// TIA Portal V18 export
DATA_BLOCK "Function Flush"   // DB47
{ S7_Optimized_Access := 'TRUE' }
VERSION : 0.1
// stored: AutoNumber true, DBAccessibleFromOPCUA true, IsOnlyStoredInLoadMemory false, IsRetainMemResEnabled false, IsWriteProtectedInAS false, MemoryReserve 100
   VAR RETAIN
      Selection : Int;
      "Input A" : Struct
         "set qty" : Real;
         "set flowrate" : Real;
         "Set time" : Int;
         "set time IN MINUTES" : Real;
         "set time in sec" : DInt;
      END_STRUCT;
      "Input B" : Struct
         "set qty" : Real;
         "set flowrate" : Real;
         "Set time" : Int;
         "set time IN MINUTES" : Real;
         "set time in sec" : DInt;
      END_STRUCT;
   END_VAR
   VAR
      "Control A" : Struct
         "Start flushing" : Bool;
         "Stop Flushing" : Bool;
         "flush running" : Bool;
         "flush Completed" : Bool;
      END_STRUCT;
      "Control B" : Struct
         "Start flushing" : Bool;
         "Stop Flushing" : Bool;
         "flush running" : Bool;
         "flush Completed" : Bool;
      END_STRUCT;
      "Output A" : Struct
         "ON pump" : Bool;
         "Running time" : Int;
         "ON  outlet Valve" : Bool;
         "Volume dispensed" : Real;
         "ON_inlet A" : Bool;
      END_STRUCT;
      "Output B" : Struct
         "ON pump" : Bool;
         "Running time" : Int;
         "ON  outlet Valve" : Bool;
         "Volume dispensed" : Real;
         "ON_inlet B" : Bool;
      END_STRUCT;
   END_VAR
   VAR RETAIN
      "Set Qty" : Real;
      Flowrate : Real;
   END_VAR
   VAR
      "AD-HMI" : Struct
         "Set qty" : Real;
         "Set time" : Int;
         "Volume dispensed" : Real;
         "Run time" : Int;
         "Flowrate set" : Real;
      END_STRUCT;
   END_VAR
BEGIN
END_DATA_BLOCK
